FUNCTION_BLOCK PUBL_105_DRILLING-ROUND_HOLE (* 105-variable local group publisher for drilling a round_hole *)
  (* Standard: 61499-2 *)
  (* Version 1.0, 21-03-12, GASR, Universidade do Estado de Santa Catarina *)
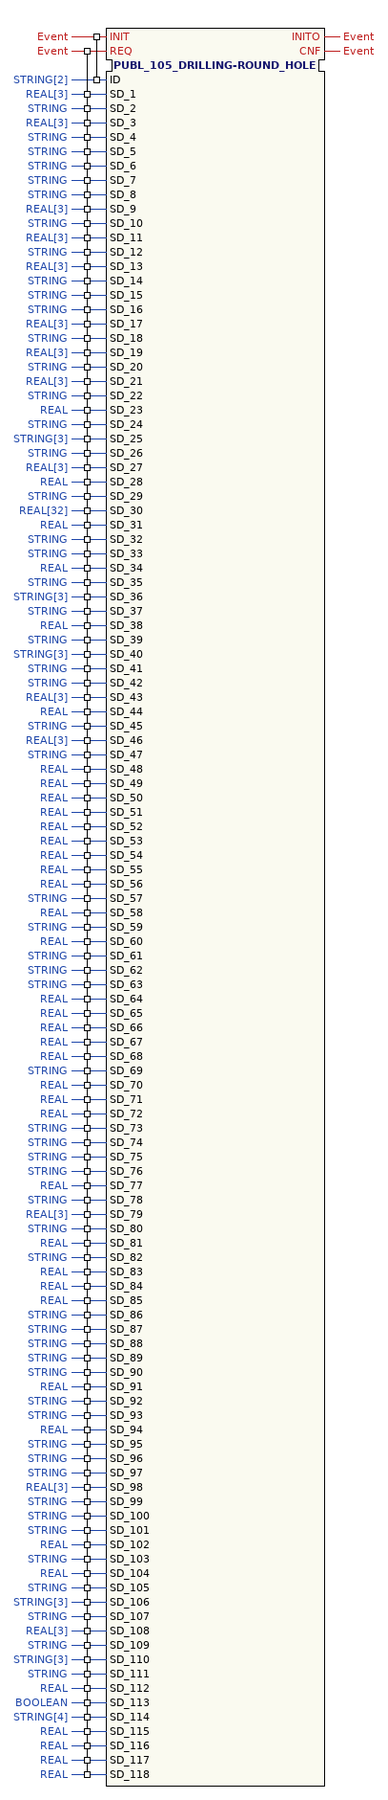
  EVENT_INPUT
    INIT WITH ID; (* Service Initialization *)
    REQ WITH SD_1, SD_2, SD_3, SD_4, SD_5, SD_6, SD_7, SD_8, SD_9, SD_10, SD_11, SD_12, SD_13, SD_14, SD_15, SD_16, SD_17, SD_18, SD_19, SD_20, SD_21, SD_22, SD_23, SD_24, SD_25, SD_26, SD_27, SD_28, SD_29, SD_30, SD_31, SD_32, SD_33, SD_34, SD_35, SD_36, SD_37, SD_38, SD_39, SD_40, SD_41, SD_42, SD_43, SD_44, SD_45, SD_46, SD_47, SD_48, SD_49, SD_50, SD_51, SD_52, SD_53, SD_54, SD_55, SD_56, SD_57, SD_58, SD_59, SD_60, SD_61, SD_62, SD_63, SD_64, SD_65, SD_66, SD_67, SD_68, SD_69, SD_70, SD_71, SD_72, SD_73, SD_74, SD_75, SD_76, SD_77, SD_78, SD_79, SD_80, SD_81, SD_82, SD_83, SD_84, SD_85, SD_86, SD_87, SD_88, SD_89, SD_90, SD_91, SD_92, SD_93, SD_94, SD_95, SD_96, SD_97, SD_98, SD_99, SD_100, SD_101, SD_102, SD_103, SD_104, SD_105, SD_106, SD_107, SD_108, SD_109, SD_110, SD_111, SD_112, SD_113, SD_114, SD_115, SD_116, SD_117, SD_118; (* Service Request *)
  END_EVENT
  EVENT_OUTPUT
    INITO; (* Initialization Confirm *)
    CNF; (* Service Confirmation *)
  END_EVENT
  VAR_INPUT
    ID : ARRAY [0..1] OF STRING; (* Default id is the FB instance name *)
    SD_1 : ARRAY [0..2] OF REAL; (* pos *)
    SD_2 : STRING; (* current_tool *)
    SD_3 : ARRAY [0..2] OF REAL; (* setup.Its_secplane.position.location.coordinates *)
    SD_4 : STRING; (* slot.its_id *)
    SD_5 : STRING; (* its_workpiece.its_id *)
    SD_6 : STRING; (* its_operations.its_id LIST - the list is concatenated in one string *)
    SD_7 : STRING; (* feature_placement.name *)
    SD_8 : STRING; (* feature_placement.location.name *)
    SD_9 : ARRAY [0..2] OF REAL; (* feature_placement.location.coordinates *)
    SD_10 : STRING; (* feature_placement.axis.its_id *)
    SD_11 : ARRAY [0..2] OF REAL; (* feature_placement.axis.direction_ratios *)
    SD_12 : STRING; (* feature_placement.ref_direction.its_id *)
    SD_13 : ARRAY [0..2] OF REAL; (* feature_placement.ref_direction_ratios *)
    SD_14 : STRING; (* depth.name *)
    SD_15 : STRING; (* depth.position.name *)
    SD_16 : STRING; (* depth.position.location.name *)
    SD_17 : ARRAY [0..2] OF REAL; (* depth.position.location.coordinates *)
    SD_18 : STRING; (* depth.position.axis.its_id *)
    SD_19 : ARRAY [0..2] OF REAL; (* depth.position.axis.direction_ratios *)
    SD_20 : STRING; (* depth.position.ref_direction.its_id *)
    SD_21 : ARRAY [0..2] OF REAL; (* depth.position.ref_direction_ratios *)
    SD_22 : STRING; (* course_of_travel *)
    SD_23 : REAL; (* course_of_travel.var1.theoretical_size *)
    SD_24 : STRING; (* course_of_travel.var1.implicit_tolerance *)
    SD_25 : ARRAY [0..2] OF STRING; (* course_of_travel.var1.{vector}, vector = {upper_limit, lower_limit, significant_digits} or {deviation,grade,its_fitting_type} *)
    SD_26 : STRING; (* course_of_travel.direction.its_id *)
    SD_27 : ARRAY [0..2] OF REAL; (* course_of_travel.direction.direction_ratios *)
    SD_28 : REAL; (* course_of_travel.sweep_angle *)
    SD_29 : STRING; (* swept_shape *)
    SD_30 : ARRAY [0..31] OF REAL; (* swept_shape.variable list *)
    SD_31 : REAL; (* swept_shape.profile_length.its_parameter_value *)
    SD_32 : STRING; (* swept_shape.profile_length.its_parameter_unit *)
    SD_33 : STRING; (* end_condition[1] *)
    SD_34 : REAL; (* end_condition[1].var1.theoretical_size *)
    SD_35 : STRING; (* end_condition[1].var1.implicit_tolerance *)
    SD_36 : ARRAY [0..2] OF STRING; (* end_condition[1].var1.{vector}, vector = {upper_limit, lower_limit, significant_digits} or {deviation,grade,its_fitting_type} *)
    SD_37 : STRING; (* end_condition[2] *)
    SD_38 : REAL; (* end_condition[2].var1.theoretical_size *)
    SD_39 : STRING; (* end_condition[2].var1.implicit_tolerance *)
    SD_40 : ARRAY [0..2] OF STRING; (* end_condition[2].var1.{vector}, vector = {upper_limit, lower_limit, significant_digits} or {deviation,grade,its_fitting_type} *)
    SD_41 : STRING; (* bottom_and_side_rough_milling.its_id *)
    SD_42 : STRING; (* its_toolpath.its_list *)
    SD_43 : ARRAY [0..2] OF REAL; (* its_tool_direction *)
    SD_44 : REAL; (* retract_plane *)
    SD_45 : STRING; (* start_point.name *)
    SD_46 : ARRAY [0..2] OF REAL; (* start_point.coordinates *)
    SD_47 : STRING; (* its_tool.its_id *)
    SD_48 : REAL; (* its_tool.its_tool_body.dimension.diameter *)
    SD_49 : REAL; (* its_tool.its_tool_body.dimension.tool_tip_half_angle *)
    SD_50 : REAL; (* its_tool.its_tool_body.dimension.tool_circumference_angle *)
    SD_51 : REAL; (* its_tool.its_tool_body.dimension.cutting_edge_lenght *)
    SD_52 : REAL; (* its_tool.its_tool_body.dimension.edge_radius *)
    SD_53 : REAL; (* its_tool.its_tool_body.dimension.edge_center_vertical *)
    SD_54 : REAL; (* its_tool.its_tool_body.dimension.edge_center_horizontal *)
    SD_55 : REAL; (* its_tool.its_tool_body.number_of_teeth *)
    SD_56 : REAL; (* its_tool.its_tool_body.hand_of_cut *)
    SD_57 : STRING; (* its_tool.its_tool_body.coolant_through *)
    SD_58 : REAL; (* its_tool.its_tool_body.pilot_length *)
    SD_59 : STRING; (* its_tool.its_tool_body.{other_tool_body_parameter} *)
    SD_60 : REAL; (* its_tool.its_cutting_edge.tool_offset_length *)
    SD_61 : STRING; (* its_tool.its_cutting_edge.its_material.standaSD_identifier *)
    SD_62 : STRING; (* its_tool.its_cutting_edge.its_material.material_identifier *)
    SD_63 : STRING; (* its_tool.its_cutting_edge.its_material.material_property.{list_of_parameters} *)
    SD_64 : REAL; (* its_tool.its_cutting_edge.its_technological_data.cutting_angle *)
    SD_65 : REAL; (* its_tool.its_cutting_edge.its_technological_data.free_angle *)
    SD_66 : REAL; (* its_tool.its_cutting_edge.its_technological_data.aux_angle *)
    SD_67 : REAL; (* its_tool.its_cutting_edge.expected_tool_life *)
    SD_68 : REAL; (* its_tool.its_cutting_edge.its_technology.feedrate *)
    SD_69 : STRING; (* its_tool.its_cutting_edge.its_technology.feedrate_reference *)
    SD_70 : REAL; (* its_tool.its_cutting_edge.its_technology.cutspeed *)
    SD_71 : REAL; (* its_tool.its_cutting_edge.its_technology.spindle *)
    SD_72 : REAL; (* its_tool.its_cutting_edge.its_technology.feedrate_per_tooth *)
    SD_73 : STRING; (* its_tool.its_cutting_edge.its_technology.sincronize_spindle_with_feed *)
    SD_74 : STRING; (* its_tool.its_cutting_edge.its_technology.inhibit_feedrate_override *)
    SD_75 : STRING; (* its_tool.its_cutting_edge.its_technology.inhibit_spindle_override *)
    SD_76 : STRING; (* its_tool.its_cutting_edge.its_technology.its_adaptive_control *)
    SD_77 : REAL; (* its_tool.overall_assembly_length *)
    SD_78 : STRING; (* its_tool.direction_for_spindle_orientation.its_id *)
    SD_79 : ARRAY [0..2] OF REAL; (* its_tool.direction_for_spindle_orientation.direction_ratios *)
    SD_80 : STRING; (* its_tool.tool_holder_diameter_for_spindle_orientation *)
    SD_81 : REAL; (* its_technology.feedrate *)
    SD_82 : STRING; (* its_technology.feedrate_reference *)
    SD_83 : REAL; (* its_technology.cutspeed *)
    SD_84 : REAL; (* its_technology.spindle *)
    SD_85 : REAL; (* its_technology.feedrate_per_tooth *)
    SD_86 : STRING; (* its_technology.sincronize_spindle_with_feed *)
    SD_87 : STRING; (* its_technology.inhibit_feedrate_override *)
    SD_88 : STRING; (* its_technology.inhibit_spindle_override *)
    SD_89 : STRING; (* its_technology.its_adaptive_control *)
    SD_90 : STRING; (* its_machine_functions.coolant *)
    SD_91 : REAL; (* its_machine_functions.coolant_pressure *)
    SD_92 : STRING; (* its_machine_functions.mist *)
    SD_93 : STRING; (* its_machine_functions.through_spindle_coolant *)
    SD_94 : REAL; (* its_machine_functions.through_pressure *)
    SD_95 : STRING; (* its_machine_functions.axis_clamping *)
    SD_96 : STRING; (* its_machine_functions.chip_removal *)
    SD_97 : STRING; (* its_machine_functions.oriented_spindle_stop.its_id *)
    SD_98 : ARRAY [0..2] OF REAL; (* its_machine_functions.oriented_spindle_stop.direction_ratios *)
    SD_99 : STRING; (* its_machine_functions.its_process_model.ini_data_file *)
    SD_100 : STRING; (* its_machine_functions.its_process_model.its_type *)
    SD_101 : STRING; (* its_machine_functions.other_functions *)
    SD_102 : REAL; (* overcut_length *)
    SD_103 : STRING; (* approach.tool_orientation.its_id *)
    SD_104 : REAL; (* approach.tool_orientation.direction_ratios *)
    SD_105 : STRING; (* approach.approach_retract_strategy (name of it) *)
    SD_106 : ARRAY [0..2] OF STRING; (* approach.approach_retract_strategy.list of parameters *)
    SD_107 : STRING; (* retract.tool_orientation.its_id *)
    SD_108 : ARRAY [0..2] OF REAL; (* retract.tool_orientation.direction_ratios *)
    SD_109 : STRING; (* retract.approach_retract_strategy (name of it) *)
    SD_110 : ARRAY [0..2] OF STRING; (* retract.approach_retract_strategy.list of parameters *)
    SD_111 : STRING; (* its_machining_strategy *)
    SD_112 : REAL; (* its_machining_strategy.overlap *)
    SD_113 : BOOLEAN; (* its_machining_strategy.allow_multiple_passes *)
    SD_114 : ARRAY [0..3] OF STRING; (* its_machining_strategy.list of parameters *)
    SD_115 : REAL; (* axial_cutting_depth *)
    SD_116 : REAL; (* radial_cutting_depth *)
    SD_117 : REAL; (* allowance_side *)
    SD_118 : REAL; (* allowance_bottom *)
  END_VAR
  SERVICE PUBL_118/SUBL_118 (* Data publication service *)
    SEQUENCE normal_establishment
      PUBL_118.INIT(ID) -> SUBL_118.INITO();
      SUBL_118.INIT(ID) -> SUBL_118.INITO();
    END_SEQUENCE
    SEQUENCE normal_data_transfer
      PUBL_118.REQ(SD_1,SD_2,SD_3,SD_4,SD_5,SD_6,SD_7,SD_8,SD_9,SD_10,SD_11,SD_12,SD_13,SD_14,SD_15,SD_16,SD_17,SD_18,SD_19,SD_20,SD_21,SD_22,SD_23,SD_24,SD_25,SD_26,SD_27,SD_28,SD_29,SD_30,SD_31,SD_32,SD_33,SD_34,SD_35,SD_36,SD_37,SD_38,SD_39,SD_40,SD_41,SD_42,SD_43,SD_44,SD_45,SD_46,SD_47,SD_48,SD_49,SD_50,SD_51,SD_52,SD_53,SD_54,SD_55,SD_56,SD_57,SD_58,SD_59,SD_60,SD_61,SD_62,SD_63,SD_64,SD_65,SD_66,SD_67,SD_68,SD_69,SD_70,SD_71,SD_72,SD_73,SD_74,SD_75,SD_76,SD_77,SD_78,SD_79,SD_80,SD_81,SD_82,SD_83,SD_84,SD_85,SD_86,SD_87,SD_88,SD_89,SD_90,SD_91,SD_92,SD_93,SD_94,SD_95,SD_96,SD_97,SD_98,SD_99,SD_100,SD_101,SD_102,SD_103,SD_104,SD_105,SD_106,SD_107,SD_108,SD_109,SD_110,SD_111,SD_112,SD_113,SD_114,SD_115,SD_116,SD_117,SD_118) -> SUBL_118.IND(RD_1,RD_2,RD_3,RD_4,RD_5,RD_6,RD_7,RD_8,RD_9,RD_10,RD_11,RD_12,RD_13,RD_14,RD_15,RD_16,RD_17,RD_18,RD_19,RD_20,RD_21,RD_22,RD_23,RD_24,RD_25,RD_26,RD_27,RD_28,RD_29,RD_30,RD_31,RD_32,RD_33,RD_34,RD_35,RD_36,RD_37,RD_38,RD_39,RD_40,RD_41,RD_42,RD_43,RD_44,RD_45,RD_46,RD_47,RD_48,RD_49,RD_50,RD_51,RD_52,RD_53,RD_54,RD_55,RD_56,RD_57,RD_58,RD_59,RD_60,RD_61,RD_62,RD_63,RD_64,RD_65,RD_66,RD_67,RD_68,RD_69,RD_70,RD_71,RD_72,RD_73,RD_74,RD_75,RD_76,RD_77,RD_78,RD_79,RD_80,RD_81,RD_82,RD_83,RD_84,RD_85,RD_86,RD_87,RD_88,RD_89,RD_90,RD_91,RD_92,RD_93,RD_94,RD_95,RD_96,RD_97,RD_98,RD_99,RD_100,RD_101,RD_102,RD_103,RD_104,RD_105,RD_106,RD_107,RD_108,RD_109,RD_110,RD_111,RD_112,RD_113,RD_114,RD_115,RD_116,RD_117,RD_118);
    END_SEQUENCE
  END_SERVICE
END_FUNCTION_BLOCK
